Staubli VAL3: JointTrajPtMsg.pjx

Parameters version=s7.7.2 stackSize=5000 millimeterUnit=true
Program file=start.pgx
Program file=stop.pgx
Data file=JointTrajPtMsg.dtx
Type name=Body path=../Body/Body.pjx
Type name=Header path=../Header/Header.pjx
Type name=Prefix path=../Prefix/Prefix.pjx
Type name=JointTrajPt path=../JointTrajPt/JointTrajPt.pjx
